{attribute 'qualified_only'}
VAR_GLOBAL
	AvvioMotore: BOOL;
	ArrestoMotore: BOOL;
	MotoreInMarcia: BOOL;
END_VAR

(* stored: Version 1.1.0.1, ProductVersion 3.1.4024.12
   GVL GVL: Id {d416722d-e6df-4566-b345-7a4655b4e1bd} *)
